{attribute 'qualified_only'}
VAR_GLOBAL
	nCylPos : INT; 
	nWinchEncoder : INT; 
	PressureSensorVals : ST_PressureSensor; 
	BoxVariables : ST_BoxParams; 
END_VAR

(* stored: Version 1.1.0.1, ProductVersion 3.1.4024.12
   GVL G_Inputs: Id {e6e68996-dfb9-4405-83ee-7cca160370dd} *)
